{attribute 'pack_mode' := '1'}
TYPE ControllerStatus EXTENDS OutgoingMessage :
STRUCT
	commLinkStatus: STRING(CT.STATUS_STRING_SIZE);
	motionEnabled: BOOL;
	lastCommandStatus: STRING(CT.STATUS_STRING_SIZE);
END_STRUCT
END_TYPE

(* stored: Version 1.1.0.1, ProductVersion 3.1.4022.12
   DUT ControllerStatus: Id {e141c568-d961-40c2-bf86-98c0e5cf1ef6} *)
